INTERFACE I_PositionalDrive EXTENDS I_Drive

PROPERTY CurrentPosition : LREAL
GET
END_GET
END_PROPERTY

METHOD ABSTRACT moveAbsolute : BOOL
VAR_INPUT
	newTarget : LREAL; 
END_VAR
END_METHOD

METHOD ABSTRACT moveRelative : BOOL
VAR_INPUT
	distance : LREAL;
END_VAR
END_METHOD

METHOD setPosition : BOOL
VAR_INPUT
	newPosition : LREAL;
END_VAR
END_METHOD

PROPERTY TargetPosition : LREAL
GET
END_GET
END_PROPERTY

END_INTERFACE

(* stored: Version 1.1.0.1, ProductVersion 3.1.4024.11
   Itf I_PositionalDrive: Id {7ff36782-3a74-44fe-9781-bd1eb4fd6a04}
   Folder Properties: Id {9fdc7af2-f2cc-46a5-9f69-d70ee615a965}
   Property CurrentPosition: Id {7bb2ba01-3d78-4401-8f5b-3022e94c3d56}
   Get Get: Id {1b8d0303-30f3-4b27-838f-974d7c0d43e7}
   Method moveAbsolute: Id {981b32ef-beee-4f5d-8a5f-d267261dbe18}
   Method moveRelative: Id {8494ae18-19d0-47fb-9dc9-c2631eaabe77}
   Method setPosition: Id {9e396a0e-8091-4d22-a167-fdf3744c0aff}
   Property TargetPosition: Id {b043ed3a-6d53-44a1-a250-c5f98bdd7456}
   Get Get: Id {7a0ab4e3-037c-47ad-b9f8-c95c28950d23} *)
